// TIA Portal V16 export
// export: Created 2022-11-17T15:49:46.6411153Z, ExportSetting WithDefaults, DisplayName Totally Integrated Automation Portal, DisplayVersion V16 Update 6, DisplayName TIA Portal Version Control Interface, DisplayVersion V16 Update 2, DisplayName TIA Portal Openness, DisplayVersion V16 Update 6, DisplayName SINAMICS Startdrive Advanced, DisplayVersion V16 Update 5, DisplayName SINAMICS Startdrive G130, G150, S120, S150, SINAMICS MV, S210, DisplayVersion V16 Update 5, DisplayName SINAMICS Startdrive G110M, G120, G120C, G120D, G120P, G115D, DisplayVersion V16 Update 5, DisplayName STEP 7 Professional, DisplayVersion V16 Update 6, DisplayName STEP 7 Safety, DisplayVersion V16, DisplayName WinCC Advanced, DisplayVersion V16 Update 6
DATA_BLOCK "DB250_ProgramData"   // DB250
{ S7_Optimized_Access := 'FALSE' }
AUTHOR : Robopac
VERSION : 0.0
// stored: AutoNumber false, IsOnlyStoredInLoadMemory false, IsWriteProtectedInAS false
   VAR RETAIN
      Program { S7_SetPoint := 'True'} : "DatiProgramma";
   END_VAR
BEGIN
   Program.Wrapping := TRUE;
   Program.TopLenght := 500;
   Program.TopRelease := 0;
   Program.TopDown := 0;
   Program.Top := 4;
   Program.PressurePTime := 0;
   Program.LifterTime := 0;
   Program.RevOverContrast := 1;
   Program.RopeEndCycle := 16#02;
   Program.Spare4 := 16#01;
   Program.RopeTime := 1500;
   Program.RevOverClamp := 1;
   Program.FilmForceFinalRev := 10;
   Program.FilmPrestretchFinalRev := 100;
   Program.ArmSpeed := 100;
   Program.CarriageDown4Top := 500;
   Program.TopDownTime := 1500;
   Program.LapsUnderTop := 0;
   Program.Spare6 := 0;
   Program.Spare7 := 0;
   Program.Spare8 := 0;
   Program.Spare9 := 0;
   Program.Spare10 := 0;
   Program.Spare11 := 0;
   Program.Spare12 := 0;
   Program.Overlap0_1 := 0;
   Program.Height1 := 130;
   Program.Landmark1 := FALSE;
   Program.Lifter1 := FALSE;
   Program.SpareBit1H1 := FALSE;
   Program.Airblower1 := TRUE;
   Program.NextStep1 := TRUE;
   Program.PressureP1 := TRUE;
   Program.SpareByte2H1 := 16#00;
   Program.Revolution1 := 1;
   Program.RopeUnit1_1 := 16#01;
   Program.RopeUnit1_2 := 16#01;
   Program.FilmForce1 := 5;
   Program.FilmPrestretch1 := 200;
   Program.Spare3H1 := 0;
   Program.Spare49 := 0;
   Program.Spare50 := 0;
   Program.Spare51 := 0;
   Program.Spare52 := 0;
   Program.Spare53 := 0;
   Program.Overlap1_2 := 0;
   Program.Height2 := 50;
   Program.Landmark2 := FALSE;
   Program.Lifter2 := FALSE;
   Program.SpareBit1H2 := FALSE;
   Program.Airblower2 := TRUE;
   Program.NextStep2 := TRUE;
   Program.PressureP2 := TRUE;
   Program.SpareByte2H2 := 16#00;
   Program.Revolution2 := 1;
   Program.RopeUnit2_1 := 16#01;
   Program.RopeUnit2_2 := 16#01;
   Program.FilmForce2 := 20;
   Program.FilmPrestretch2 := 200;
   Program.Spare3H2 := 0;
   Program.Spare54 := 0;
   Program.Spare55 := 0;
   Program.Spare56 := 0;
   Program.Spare57 := 0;
   Program.Spare58 := 0;
   Program.Overlap2_3 := 100;
   Program.Height3 := -50;
   Program.Landmark3 := TRUE;
   Program.Lifter3 := FALSE;
   Program.SpareBit1H3 := FALSE;
   Program.Airblower3 := TRUE;
   Program.NextStep3 := TRUE;
   Program.PressureP3 := TRUE;
   Program.SpareByte2H3 := 16#00;
   Program.Revolution3 := 2;
   Program.RopeUnit3_1 := 16#01;
   Program.RopeUnit3_2 := 16#01;
   Program.FilmForce3 := 30;
   Program.FilmPrestretch3 := 200;
   Program.Spare3H3 := 0;
   Program.Spare59 := 0;
   Program.Spare60 := 0;
   Program.Spare61 := 380;
   Program.Spare62 := 2800;
   Program.Spare63 := 0;
   Program.Overlap3_4 := 100;
   Program.Height4 := 100;
   Program.Landmark4 := FALSE;
   Program.Lifter4 := FALSE;
   Program.SpareBit1H4 := FALSE;
   Program.Airblower4 := TRUE;
   Program.NextStep4 := TRUE;
   Program.PressureP4 := TRUE;
   Program.SpareByte2H4 := 16#00;
   Program.Revolution4 := 3;
   Program.RopeUnit4_1 := 16#02;
   Program.RopeUnit4_2 := 16#02;
   Program.FilmForce4 := 30;
   Program.FilmPrestretch4 := 200;
   Program.Spare3H4 := 0;
   Program.Spare64 := 0;
   Program.Spare65 := 0;
   Program.Spare66 := 0;
   Program.Spare67 := 0;
   Program.Spare68 := 0;
   Program.Overlap4_5 := 0;
   Program.Height5 := 50;
   Program.Landmark5 := FALSE;
   Program.Lifter5 := FALSE;
   Program.SpareBit1H5 := FALSE;
   Program.Airblower5 := TRUE;
   Program.NextStep5 := FALSE;
   Program.PressureP5 := FALSE;
   Program.SpareByte2H5 := 16#00;
   Program.Revolution5 := 1;
   Program.RopeUnit5_1 := 16#01;
   Program.RopeUnit5_2 := 16#01;
   Program.FilmForce5 := 30;
   Program.FilmPrestretch5 := 200;
   Program.Spare3H5 := 0;
   Program.Spare69 := 0;
   Program.Spare70 := 0;
   Program.Spare71 := 0;
   Program.Spare72 := 0;
   Program.Spare73 := 0;
   Program.Overlap5_6 := 100;
   Program.Height6 := 50;
   Program.Landmark6 := FALSE;
   Program.Lifter6 := FALSE;
   Program.SpareBit1H6 := FALSE;
   Program.Airblower6 := TRUE;
   Program.NextStep6 := FALSE;
   Program.PressureP6 := FALSE;
   Program.SpareByte2H6 := 16#00;
   Program.Revolution6 := 2;
   Program.RopeUnit6_1 := 16#02;
   Program.RopeUnit6_2 := 16#01;
   Program.FilmForce6 := 20;
   Program.FilmPrestretch6 := 200;
   Program.Spare3H6 := 0;
   Program.Spare74 := 0;
   Program.Spare75 := 0;
   Program.Spare76 := 0;
   Program.Spare77 := 0;
   Program.Spare78 := 0;
   Program.Overlap6_7 := 0;
   Program.Height7 := 0;
   Program.Landmark7 := FALSE;
   Program.Lifter7 := FALSE;
   Program.SpareBit1H7 := FALSE;
   Program.Airblower7 := FALSE;
   Program.NextStep7 := TRUE;
   Program.PressureP7 := FALSE;
   Program.SpareByte2H7 := 16#00;
   Program.Revolution7 := 1;
   Program.RopeUnit7_1 := 16#01;
   Program.RopeUnit7_2 := 16#01;
   Program.FilmForce7 := 0;
   Program.FilmPrestretch7 := 100;
   Program.Spare3H7 := 0;
   Program.Spare79 := 0;
   Program.Spare80 := 0;
   Program.Spare81 := 0;
   Program.Spare82 := 0;
   Program.Spare83 := 0;
   Program.Overlap7_8 := 0;
   Program.Height8 := 0;
   Program.Landmark8 := FALSE;
   Program.Lifter8 := FALSE;
   Program.SpareBit1H8 := FALSE;
   Program.Airblower8 := FALSE;
   Program.NextStep8 := TRUE;
   Program.PressureP8 := FALSE;
   Program.SpareByte2H8 := 16#00;
   Program.Revolution8 := 1;
   Program.RopeUnit8_1 := 16#01;
   Program.RopeUnit8_2 := 16#01;
   Program.FilmForce8 := 0;
   Program.FilmPrestretch8 := 100;
   Program.Spare3H8 := 0;
   Program.Spare84 := 0;
   Program.Spare85 := 0;
   Program.Spare86 := 0;
   Program.Spare87 := 0;
   Program.Spare88 := 0;
   Program.Overlap8_9 := 0;
   Program.Height9 := 0;
   Program.Landmark9 := FALSE;
   Program.Lifter9 := FALSE;
   Program.SpareBit1H9 := FALSE;
   Program.Airblower9 := FALSE;
   Program.NextStep9 := TRUE;
   Program.PressureP9 := FALSE;
   Program.SpareByte2H9 := 16#00;
   Program.Revolution9 := 1;
   Program.RopeUnit9_1 := 16#01;
   Program.RopeUnit9_2 := 16#01;
   Program.FilmForce9 := 0;
   Program.FilmPrestretch9 := 100;
   Program.Spare3H9 := 0;
   Program.Spare89 := 0;
   Program.Spare90 := 0;
   Program.Spare91 := 0;
   Program.Spare92 := 0;
   Program.Spare93 := 0;
   Program.Overlap9_10 := 0;
   Program.Height10 := 0;
   Program.Landmark10 := FALSE;
   Program.Lifter10 := FALSE;
   Program.SpareBit1H10 := FALSE;
   Program.Airblower10 := FALSE;
   Program.NextStep10 := FALSE;
   Program.PressureP10 := FALSE;
   Program.SpareByte2H10 := 16#00;
   Program.Revolution10 := 1;
   Program.RopeUnit10_1 := 16#01;
   Program.RopeUnit10_2 := 16#01;
   Program.FilmForce10 := 0;
   Program.FilmPrestretch10 := 100;
   Program.Spare3H10 := 0;
   Program.Spare94 := 0;
   Program.Spare95 := 0;
   Program.Spare96 := 0;
   Program.Spare97 := 0;
   Program.Spare98 := 0;
   Program.Overlap10_11 := 0;
   Program.Height11 := 0;
   Program.Landmark11 := FALSE;
   Program.Lifter11 := FALSE;
   Program.SpareBit1H11 := FALSE;
   Program.Airblower11 := FALSE;
   Program.NextStep11 := TRUE;
   Program.PressureP11 := FALSE;
   Program.SpareByte2H11 := 16#00;
   Program.Revolution11 := 1;
   Program.RopeUnit11_1 := 16#01;
   Program.RopeUnit11_2 := 16#01;
   Program.FilmForce11 := 0;
   Program.FilmPrestretch11 := 100;
   Program.Spare3H11 := 0;
   Program.Spare99 := 0;
   Program.Spare100 := 0;
   Program.Spare101 := 0;
   Program.Spare102 := 0;
   Program.Spare103 := 0;
   Program.Overlap11_12 := 0;
   Program.Height12 := 0;
   Program.Landmark12 := FALSE;
   Program.Lifter12 := FALSE;
   Program.SpareBit1H12 := FALSE;
   Program.Airblower12 := FALSE;
   Program.NextStep12 := FALSE;
   Program.PressureP12 := FALSE;
   Program.SpareByte2H12 := 16#00;
   Program.Revolution12 := 1;
   Program.RopeUnit12_1 := 16#01;
   Program.RopeUnit12_2 := 16#01;
   Program.FilmForce12 := 0;
   Program.FilmPrestretch12 := 100;
   Program.Spare3H12 := 0;
   Program.Spare104 := 0;
   Program.Spare105 := 0;
   Program.Spare106 := 0;
   Program.Spare107 := 0;
   Program.Spare108 := 0;
END_DATA_BLOCK
